PROGRAM MAIN
VAR
END_VAR

END_PROGRAM

(* stored: Version 1.1.0.1
   POU MAIN: Id {5a07e6d0-257c-4939-8426-e926921b8031} *)
